{attribute 'strict'}
TYPE E_VisionJob :
(
	CASE_RECEIVER_E25_0100812762 := 0
);
END_TYPE

(* stored: Version 1.1.0.1, ProductVersion 3.1.4024.9
   DUT E_VisionJob: Id {c15c3b8c-9186-4696-9e1d-0ee705d2c942} *)
